Staubli VAL3: ChangeLength.pgx

public program ChangeLength(pointRx& x_trSource[], num& x_nLength[])
  local num l_nBuff[2]
begin


  //参数合法化处理
  if size(x_trSource)<3
    return
  endIf

  l_nBuff[0]=distance(x_trSource[0].trsf,x_trSource[1].trsf)
  l_nBuff[1]=distance(x_trSource[2].trsf,x_trSource[1].trsf)


  if x_nLength[1]<=0 or x_nLength[0]<=0 or l_nBuff[0]<=0 or l_nBuff[1]<=0
    return
  endIf



  x_trSource[0].trsf.x=(x_trSource[0].trsf.x-x_trSource[1].trsf.x)/l_nBuff[0]*x_nLength[0]+x_trSource[1].trsf.x
  x_trSource[0].trsf.y=(x_trSource[0].trsf.y-x_trSource[1].trsf.y)/l_nBuff[0]*x_nLength[0]+x_trSource[1].trsf.y
  x_trSource[0].trsf.z=(x_trSource[0].trsf.z-x_trSource[1].trsf.z)/l_nBuff[0]*x_nLength[0]+x_trSource[1].trsf.z

  x_trSource[2].trsf.x=(x_trSource[2].trsf.x-x_trSource[1].trsf.x)/l_nBuff[1]*x_nLength[1]+x_trSource[1].trsf.x
  x_trSource[2].trsf.y=(x_trSource[2].trsf.y-x_trSource[1].trsf.y)/l_nBuff[1]*x_nLength[1]+x_trSource[1].trsf.y
  x_trSource[2].trsf.z=(x_trSource[2].trsf.z-x_trSource[1].trsf.z)/l_nBuff[1]*x_nLength[1]+x_trSource[1].trsf.z









end
